PROGRAM couple
VAR
	mcGearIn			: MC_GearIn;
	shouldGearIn		: BOOL;
	
	mcGearOut			: MC_GearOut;
	shouldGearOut		: BOOL;
END_VAR

METHOD checkGearIn : BOOL
VAR_INPUT
END_VAR
mcGearIn(
	Master:= master.axis, 
	Slave:= slave.axis, 
	Execute:= shouldGearIn, 
	RatioNumerator:= 1, // 从轴速度
	RatioDenominator:= 1, // 主轴速度
	Acceleration:= , 
	Deceleration:= , 
	Jerk:= , 
	BufferMode:= , 
	Options:= , 
	InGear=> , 
	Busy=> , 
	Active=> , 
	CommandAborted=> , 
	Error=> , 
	ErrorID=> );
END_METHOD

METHOD checkGearOut : BOOL
VAR_INPUT
END_VAR
mcGearOut(
	Slave:= slave.axis, 
	Execute:= shouldGearOut, 
	Options:= , 
	Done=> , 
	Busy=> , 
	Error=> , 
	ErrorID=> );
END_METHOD

END_PROGRAM

(* stored: Version 1.1.0.1, ProductVersion 3.1.4024.4
   POU couple: Id {6b92097d-4e58-4a28-ae5d-24f146ac388b}, SpecialFunc None
   Method checkGearIn: Id {42c2cda4-7bfb-49a1-ac31-e31dc7e42c68}
   Method checkGearOut: Id {5e72b8e4-d3fb-4dd3-b7a0-5288e35c7e40} *)
